Universal Robots PolyScope program: rrp p1.urp

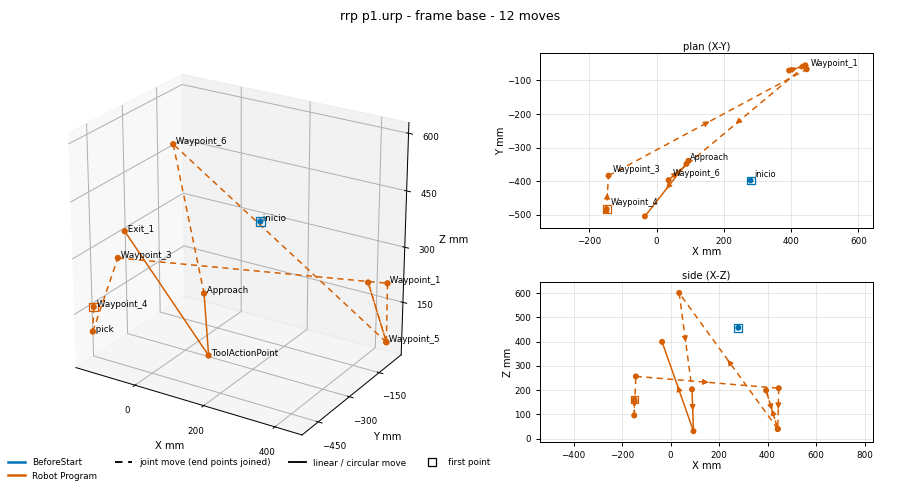
[picture p0: tool path of rrp p1.urp in frame base, 12 of 12 moves have a stored position in this frame; points joined in program order, loops and branches not executed]
Program rrp p1 (installation=default directory=/programs createdIn=5.14.5 lastSavedIn=5.14.5 robotSerialNumber=20195300809)
Calibrated DH parameters: a=[-0.000085, -0.20076, -0.212369, 0.000121, -0.000118, 0]; d=[0.15185, -26.306375, 24.753047, 1.684739, 0.085386, 0.092088]; alpha=[1.572149, -0.00522, -0.011864, 1.571339, -1.571085, 0]; deltaTheta=[0, 0.599885, -0.513355, -0.086555, 0.000006, 0]
InitVariablesNode variables(variable(name=Pallet_1_cnt_1, expression=1), variable(name=Pallet_1_lct, expression=1), variable(name=Pallet_1_lno, expression=1), variable(name=Pallet_1_sep, expression=False), variable(name=Pallet_1_tct, expression=1))
BeforeStart
  Set DigitalOutput pin=digital_out[0]; digitalValue=1
  URCap Gripper Activate (Robotiq_Grippers, Robotiq Inc.) dataModel(ResetAndActivateKey=false)
  URCap Gripper (Robotiq_Grippers, Robotiq Inc.) dataModel(position=39.6078431372549, force=0.0, speed=0.0, positionInDouble=39.6078431372549, forceInDouble=0.0, speedInDouble=0.0, slaveIds=[9], blocking=true)
  MoveJ speed 60 deg/s, acceleration 80 deg/s^2 (useActiveTCP=true) feature=Base
    Waypoint inicio: TCP in base x=279.414 y=-397.704 z=457.414 mm, rx=0.1136 ry=-2.0634 rz=2.2425 rad; joints [-0.575, -86.871, -83.093, -96.944, -5.349, 80.157] deg; TCP offset x=0 y=0 z=174 mm, rx=0 ry=0 rz=0 rad
Robot Program (runOnlyOnce=false)
  If digital_in[0]==0
    Wait Sleep waitTime=1.5
    Set DigitalOutput pin=digital_out[0]; digitalValue=0
    MoveJ speed 60 deg/s, acceleration 80 deg/s^2 (useActiveTCP=true) feature=Base
      Waypoint Waypoint_4: TCP in base x=-148.929 y=-482.772 z=161.199 mm, rx=2.2066 ry=2.1401 rz=-0.1444 rad; joints [-91.68, -146.455, 4.446, -121.567, 88.128, 90.699] deg
      Waypoint pick: TCP in base x=-149.946 y=-488.344 z=95.513 mm, rx=2.2157 ry=2.2135 rz=-0.0641 rad; joints [-91.736, -141.984, -22.125, -103.826, 87.948, 88.828] deg; TCP offset x=0 y=0 z=174 mm, rx=0 ry=0 rz=0 rad
      URCap Gripper (Robotiq_Grippers, Robotiq Inc.) dataModel(position=100.0, force=30.0, speed=100.0, positionInDouble=100.0, forceInDouble=30.0, speedInDouble=100.0, slaveIds=[9], blocking=true)
      Waypoint Waypoint_3: TCP in base x=-143.244 y=-383.342 z=256.79 mm, rx=-0.001 ry=-3.1198 rz=0.1382 rad; joints [-91.408, -126.47, -1.653, -136.781, 88.514, -0.559] deg; TCP offset x=0 y=0 z=174 mm, rx=0 ry=0 rz=0 rad
      Waypoint Waypoint_1: TCP in base x=446.334 y=-66.794 z=207.968 mm, rx=-2.2031 ry=2.1153 rz=-0.1526 rad; joints [9.174, -120.095, -31.916, -110.723, 87.614, 7.353] deg
      Waypoint Waypoint_5: TCP in base x=442.284 y=-55.675 z=39.778 mm, rx=2.2666 ry=-2.1521 rz=-0.0076 rad; joints [9.922, -124.016, -68.089, -78.783, 88.931, 7.213] deg
      URCap Gripper (Robotiq_Grippers, Robotiq Inc.) dataModel(position=39.6078431372549, force=0.0, speed=0.0, positionInDouble=39.6078431372549, forceInDouble=0.0, speedInDouble=0.0, slaveIds=[9], blocking=true)
      Waypoint Waypoint_2: TCP in base x=394.091 y=-70.578 z=198.821 mm, rx=-2.2702 ry=2.0281 rz=-0.0275 rad; joints [6.648, -107.871, -51.747, -105.478, 92.268, 0.881] deg
      Wait Sleep waitTime=2
      Waypoint Waypoint_5: TCP in base x=442.284 y=-55.675 z=39.778 mm, rx=2.2666 ry=-2.1521 rz=-0.0076 rad; joints [9.922, -124.016, -68.089, -78.783, 88.931, 7.213] deg
      URCap Gripper (Robotiq_Grippers, Robotiq Inc.) dataModel(position=100.0, force=0.0, speed=0.0, positionInDouble=100.0, forceInDouble=0.0, speedInDouble=0.0, slaveIds=[9], blocking=true)
      Waypoint Waypoint_6: TCP in base x=35.389 y=-396.597 z=600.979 mm, rx=0.0786 ry=-2.0734 rz=2.2118 rad; joints [-2.521, -64.815, -43.699, -155.357, -3.819, 77.412] deg; TCP offset x=0 y=0 z=174 mm, rx=0 ry=0 rz=0 rad
      URCap Palletizing (polyscope-pallet-impl, Universal Robots) dataModel(palletFeature=Base, isPalletizing=true, Variable(key=name, variable(name=Pallet_1)), Variable(key=globalCountingVariable, variable(name=Pallet_1_cnt_1, initializeExpression=1)), Variable(key=layerNumberVariable, variable(name=Pallet_1_lno, initializeExpression=1)), Variable(key=layerCountingVariable, variable(name=Pallet_1_lct, initializeExpression=1)), Variable(key=handleSeparatorVariable, variable(name=Pallet_1_sep, initializeExpression=False)), Variable(key=totalCountVariable, variable(name=Pallet_1_tct, initializeExpression=1)), Length(key=objectHeight value=0.02 unit=M), Variable(key=referencePoint, variable(featureName=referencePoint)), Variable(key=separatorPoint, variable(featureName=separatorPoint))); state(isChildrenLocked=true)
        URCap Patterns (polyscope-pallet-impl, Universal Robots) state(isChildrenLocked=true)
          URCap Pattern (polyscope-pallet-impl, Universal Robots) dataModel(UUID=3bedde3f-13ea-429a-8241-44f52d5ecffa, patternType=GRID, columns=3, rows=2, Variable(key=nameVariable, variable(name=Grid_Pattern_1))); state(isChildrenLocked=true)
            URCap Item (polyscope-pallet-impl, Universal Robots) dataModel(UUID=e43305f8-078c-420c-960d-2b8ad850342d, patternType=GRID, index=0, calibrationDeltaTheta=[2.0871938292282843E-8, 0.5998849625986696, -0.513354759222901, -0.08655474087847535, 6.239817607139875E-6, -6.658617090343766E-8], calibrationA=[-8.52060452638757E-5, -0.2007601879611388, -0.2123691625519033, 1.2105607098011576E-4, -1.1833705743435544E-4, 0.0], calibrationD=[0.15184970286177432, -26.306374840159272, 24.75304670983349, 1.6847390881089916, 0.085385969004481, 0.09208826337351553], calibrationAlpha=[1.5721487795181908, -0.005219907129425837, -0.011864150755780208, 1.5713392161993658, -1.5710853432049288, 0.0], calibrationJointChecksum=[-1860213401, -1859864814, -1494669377, -1328152407, -1329437658, -1329056899], calibrationStatus=2, calibrationValidChecksum=true, baseToFeature=[0.0, 0.0, 0.0, 0.0, 0.0, 0.0], TCPOffset=[3.181769127960643E-6, -6.629856373341347E-7, 0.17399456628949236, 8.246127819572848E-6, -1.872312838325845E-5, -3.107981324938017E-5], Variable(key=variable, variable(name=CornerItem_1)), JointPositions(key=jointpositions, JointPosition(key=[1], Angle(key=pos value=-0.909138 unit=RAD)), JointPosition(key=[2], Angle(key=pos value=-1.703851 unit=RAD)), JointPosition(key=[3], Angle(key=pos value=-1.781635 unit=RAD)), JointPosition(key=[4], Angle(key=pos value=-1.224611 unit=RAD)), JointPosition(key=[5], Angle(key=pos value=1.56217 unit=RAD)), JointPosition(key=[6], Angle(key=pos value=0.715673 unit=RAD))))
            URCap Item (polyscope-pallet-impl, Universal Robots) dataModel(UUID=a102ef56-4b88-463e-b2ec-8b6804c0a8e8, patternType=GRID, index=1, calibrationDeltaTheta=[2.0871938292282843E-8, 0.5998849625986696, -0.513354759222901, -0.08655474087847535, 6.239817607139875E-6, -6.658617090343766E-8], calibrationA=[-8.52060452638757E-5, -0.2007601879611388, -0.2123691625519033, 1.2105607098011576E-4, -1.1833705743435544E-4, 0.0], calibrationD=[0.15184970286177432, -26.306374840159272, 24.75304670983349, 1.6847390881089916, 0.085385969004481, 0.09208826337351553], calibrationAlpha=[1.5721487795181908, -0.005219907129425837, -0.011864150755780208, 1.5713392161993658, -1.5710853432049288, 0.0], calibrationJointChecksum=[-1860213401, -1859864814, -1494669377, -1328152407, -1329437658, -1329056899], calibrationStatus=2, calibrationValidChecksum=true, baseToFeature=[0.0, 0.0, 0.0, 0.0, 0.0, 0.0], TCPOffset=[4.995536074636764E-6, 8.019679097692745E-6, 0.17400212486069994, -4.984431443984701E-5, 1.666783651570184E-5, 1.6236706203037297E-5], Variable(key=variable, variable(name=CornerItem_2)), JointPositions(key=jointpositions, JointPosition(key=[1], Angle(key=pos value=-0.508868 unit=RAD)), JointPosition(key=[2], Angle(key=pos value=-2.029692 unit=RAD)), JointPosition(key=[3], Angle(key=pos value=-1.419533 unit=RAD)), JointPosition(key=[4], Angle(key=pos value=-1.201603 unit=RAD)), JointPosition(key=[5], Angle(key=pos value=1.493474 unit=RAD)), JointPosition(key=[6], Angle(key=pos value=1.094403 unit=RAD))))
            URCap Item (polyscope-pallet-impl, Universal Robots) dataModel(UUID=1bf7074b-5352-416d-83c7-ed10fc9d5543, patternType=GRID, index=2, calibrationDeltaTheta=[2.0871938292282843E-8, 0.5998849625986696, -0.513354759222901, -0.08655474087847535, 6.239817607139875E-6, -6.658617090343766E-8], calibrationA=[-8.52060452638757E-5, -0.2007601879611388, -0.2123691625519033, 1.2105607098011576E-4, -1.1833705743435544E-4, 0.0], calibrationD=[0.15184970286177432, -26.306374840159272, 24.75304670983349, 1.6847390881089916, 0.085385969004481, 0.09208826337351553], calibrationAlpha=[1.5721487795181908, -0.005219907129425837, -0.011864150755780208, 1.5713392161993658, -1.5710853432049288, 0.0], calibrationJointChecksum=[-1860213401, -1859864814, -1494669377, -1328152407, -1329437658, -1329056899], calibrationStatus=2, calibrationValidChecksum=true, baseToFeature=[0.0, 0.0, 0.0, 0.0, 0.0, 0.0], TCPOffset=[9.73938988862999E-6, 1.744025429101237E-6, 0.17400164455134903, -3.839505754792504E-5, 2.6242912679330455E-6, 3.0432825196964382E-5], Variable(key=variable, variable(name=CornerItem_3)), JointPositions(key=jointpositions, JointPosition(key=[1], Angle(key=pos value=-0.286803 unit=RAD)), JointPosition(key=[2], Angle(key=pos value=-1.798895 unit=RAD)), JointPosition(key=[3], Angle(key=pos value=-1.665451 unit=RAD)), JointPosition(key=[4], Angle(key=pos value=-1.23378 unit=RAD)), JointPosition(key=[5], Angle(key=pos value=1.519199 unit=RAD)), JointPosition(key=[6], Angle(key=pos value=1.304667 unit=RAD))))
            URCap Item (polyscope-pallet-impl, Universal Robots) dataModel(UUID=abcda0fd-094c-4e7b-bace-be37c0666e4e, patternType=GRID, index=3, calibrationDeltaTheta=[2.0871938292282843E-8, 0.5998849625986696, -0.513354759222901, -0.08655474087847535, 6.239817607139875E-6, -6.658617090343766E-8], calibrationA=[-8.52060452638757E-5, -0.2007601879611388, -0.2123691625519033, 1.2105607098011576E-4, -1.1833705743435544E-4, 0.0], calibrationD=[0.15184970286177432, -26.306374840159272, 24.75304670983349, 1.6847390881089916, 0.085385969004481, 0.09208826337351553], calibrationAlpha=[1.5721487795181908, -0.005219907129425837, -0.011864150755780208, 1.5713392161993658, -1.5710853432049288, 0.0], calibrationJointChecksum=[-1860213401, -1859864814, -1494669377, -1328152407, -1329437658, -1329056899], calibrationStatus=2, calibrationValidChecksum=true, baseToFeature=[0.0, 0.0, 0.0, 0.0, 0.0, 0.0], TCPOffset=[-8.426507469017075E-6, -7.46180452962375E-6, 0.1739902854287149, 3.453387029155264E-5, -4.500722325071069E-5, 4.8910097953678515E-6], Variable(key=variable, variable(name=CornerItem_4)), JointPositions(key=jointpositions, JointPosition(key=[1], Angle(key=pos value=-0.65493 unit=RAD)), JointPosition(key=[2], Angle(key=pos value=-1.264097 unit=RAD)), JointPosition(key=[3], Angle(key=pos value=-2.211559 unit=RAD)), JointPosition(key=[4], Angle(key=pos value=-1.234987 unit=RAD)), JointPosition(key=[5], Angle(key=pos value=1.586827 unit=RAD)), JointPosition(key=[6], Angle(key=pos value=0.916658 unit=RAD))))
        URCap Layers (polyscope-pallet-impl, Universal Robots) dataModel(separators=[false], selectedPatterns=[3bedde3f-13ea-429a-8241-44f52d5ecffa])
        URCap At Each Item (polyscope-pallet-impl, Universal Robots) dataModel(selectedPattern=3bedde3f-13ea-429a-8241-44f52d5ecffa, selectedPosition=e43305f8-078c-420c-960d-2b8ad850342d, Approach_calibrationDeltaTheta=[2.0871938292282843E-8, 0.5998849625986696, -0.513354759222901, -0.08655474087847535, 6.239817607139875E-6, -6.658617090343766E-8], Approach_calibrationA=[-8.52060452638757E-5, -0.2007601879611388, -0.2123691625519033, 1.2105607098011576E-4, -1.1833705743435544E-4, 0.0], Approach_calibrationD=[0.15184970286177432, -26.306374840159272, 24.75304670983349, 1.6847390881089916, 0.085385969004481, 0.09208826337351553], Approach_calibrationAlpha=[1.5721487795181908, -0.005219907129425837, -0.011864150755780208, 1.5713392161993658, -1.5710853432049288, 0.0], Approach_calibrationJointChecksum=[-1860213401, -1859864814, -1494669377, -1328152407, -1329437658, -1329056899], Approach_calibrationStatus=2, Approach_calibrationValidChecksum=true, Approach_baseToFeature=[0.0, 0.0, 0.0, 0.0, 0.0, 0.0], Approach_TCPOffset=[-4.7305383764489894E-6, 1.3256835145358803E-5, 0.17402777380777654, -8.950663433786311E-5, 6.994195576545914E-5, -1.726397430487659E-5], Exit_calibrationDeltaTheta=[2.0871938292282843E-8, 0.5998849625986696, -0.513354759222901, -0.08655474087847535, 6.239817607139875E-6, -6.658617090343766E-8], Exit_calibrationA=[-8.52060452638757E-5, -0.2007601879611388, -0.2123691625519033, 1.2105607098011576E-4, -1.1833705743435544E-4, 0.0], Exit_calibrationD=[0.15184970286177432, -26.306374840159272, 24.75304670983349, 1.6847390881089916, 0.085385969004481, 0.09208826337351553], Exit_calibrationAlpha=[1.5721487795181908, -0.005219907129425837, -0.011864150755780208, 1.5713392161993658, -1.5710853432049288, 0.0], Exit_calibrationJointChecksum=[-1860213401, -1859864814, -1494669377, -1328152407, -1329437658, -1329056899], Exit_calibrationStatus=2, Exit_calibrationValidChecksum=true, Exit_baseToFeature=[0.0, 0.0, 0.0, 0.0, 0.0, 0.0], Exit_TCPOffset=[-1.769746453079285E-5, 1.0990106829644741E-5, 0.17400900615267095, -6.990589585355558E-5, 9.21505530727856E-6, -4.6984431037037E-5], currentWizardState=LANDING, Pose(key=refBaseToFeature, Position(key=posePosition, Length(key=X value=0 unit=M), Length(key=Y value=0 unit=M), Length(key=Z value=0 unit=M)), Rotation(key=poseRotation, Angle(key=RX value=0 unit=RAD), Angle(key=RY value=0 unit=RAD), Angle(key=RZ value=0 unit=RAD))), Pose(key=refPose, Position(key=posePosition, Length(key=X value=0.094426 unit=M), Length(key=Y value=-0.339023 unit=M), Length(key=Z value=0.030621 unit=M)), Rotation(key=poseRotation, Angle(key=RX value=0.028645 unit=RAD), Angle(key=RY value=-3.131211 unit=RAD), Angle(key=RZ value=0.009843 unit=RAD))), JointPositions(key=Approach_jointpositions, JointPosition(key=[1], Angle(key=pos value=-0.933801 unit=RAD)), JointPosition(key=[2], Angle(key=pos value=-1.743902 unit=RAD)), JointPosition(key=[3], Angle(key=pos value=-1.026665 unit=RAD)), JointPosition(key=[4], Angle(key=pos value=-1.920793 unit=RAD)), JointPosition(key=[5], Angle(key=pos value=1.534728 unit=RAD)), JointPosition(key=[6], Angle(key=pos value=0.661135 unit=RAD))), JointPositions(key=Exit_jointpositions, JointPosition(key=[1], Angle(key=pos value=-0.944849 unit=RAD)), JointPosition(key=[2], Angle(key=pos value=-1.685918 unit=RAD)), JointPosition(key=[3], Angle(key=pos value=-0.65185 unit=RAD)), JointPosition(key=[4], Angle(key=pos value=-2.316992 unit=RAD)), JointPosition(key=[5], Angle(key=pos value=1.566755 unit=RAD)), JointPosition(key=[6], Angle(key=pos value=0.595171 unit=RAD))))
          URCap Generated Movements (polyscope-pallet-impl, Universal Robots) state(isChildrenLocked=true)
            MoveJ speed 60 deg/s, acceleration 80 deg/s^2 (useActiveTCP=true) feature=referencePoint
              Waypoint Approach: TCP in base x=88.442 y=-348.461 z=203.38 mm, rx=-0.022 ry=-3.1328 rz=0.0507 rad; joints [-53.501, -99.921, -58.825, -110.055, 87.933, 37.881] deg; TCP offset x=0 y=0 z=174 mm, rx=0 ry=0 rz=0 rad; feature pose in base x=94.426 y=-339.023 z=30.621 mm, rx=0.0286 ry=-3.1312 rz=0.0098 rad
            MoveL speed 250 mm/s, acceleration 1200 mm/s^2 (useActiveTCP=true) feature(featureName=referencePoint)
              Waypoint ToolActionPoint: TCP in base x=94.426 y=-339.023 z=30.621 mm, rx=0.0286 ry=-3.1312 rz=0.0098 rad; joints [-52.168, -101.482, -104.141, -64.426, 88.715, 36.85] deg; TCP offset x=-0.009 y=0.016 z=174.005 mm, rx=-0.0001 ry=0 rz=0 rad
            Folder Tool action
              URCap Gripper (Robotiq_Grippers, Robotiq Inc.) dataModel(position=39.6078431372549, force=0.0, speed=0.0, positionInDouble=39.6078431372549, forceInDouble=0.0, speedInDouble=0.0, slaveIds=[9], blocking=true)
            MoveL speed 250 mm/s, acceleration 1200 mm/s^2 (useActiveTCP=true) feature(featureName=referencePoint)
              Waypoint Exit_1: TCP in base x=-35.067 y=-504.35 z=399.172 mm, rx=-0.0491 ry=2.1665 rz=-2.1549 rad; joints [-71.207, -92.327, -109.361, 21.619, 75.915, 1.668] deg; TCP offset x=0 y=0 z=174 mm, rx=0 ry=0 rz=0 rad
      Set DigitalOutput pin=digital_out[0]; digitalValue=1
